{attribute 'GeneratedUsingTerminal: EK1100-0000-0018'}
{attribute addProperty BoxType "EK1100-0000-0018"}
{attribute addProperty Id "Beckhoff_EP3xxxEK1122Beckhoff_EP3xxxEK1122_28DAC1C92708"}
{attribute addProperty CRC "1052505260"}
{attribute addProperty Size "2708"}
TYPE Beckhoff_EP3xxx_3EBBF4AC EXTENDS EK1100_1FC0878B :
STRUCT
	{attribute addProperty Name "Beckhoff_EP3xxxEK1122"}
	{attribute addProperty PreviousPort "Beckhoff EP3xxx : B"}
	Beckhoff_EP3xxxEK1122 : Beckhoff_EP3xxxEK1122_28DAC1C9;
END_STRUCT
END_TYPE

(* stored: Version 1.2.0.0, ProductVersion 3.1.4024.9
   DUT Beckhoff_EP3xxx_3EBBF4AC: Id {5c709629-c3a1-4d62-b536-e2263949c068} *)
